TYPE ST_MYSQLConnectionInfo :
STRUCT
	user:STRING(50):='';
	password:STRING(100):='';
	server:STRING(100):='localhost';
	DB:String(50):='';
END_STRUCT
END_TYPE

(* stored: Version 1.1.0.1, ProductVersion 3.1.4024.2
   DUT ST_MYSQLConnectionInfo: Id {de25bd10-040f-4cef-b9d0-1b900bf3a613} *)
